TYPE ST_FCSLTraceMessage :
    STRUCT
        Timestamp : T_MaxString;
        Message   : T_MaxString;
		logType   : E_LogType;
        Source    : T_MaxString;
        Context   : T_MaxString;
        ScanCount : UDINT;
        Flags     : UDINT;
        Json      : T_MaxString;
    END_STRUCT
END_TYPE

(* stored: Version 1.1.0.1
   DUT ST_FCSLTraceMessage: Id {242ca52c-3daf-4921-a4c8-16e3e378d102} *)
